Fanuc KAREL source: kt00972.KL

-- PROVISIONAL review KL for V770-1; original PC SHA256 310e2f795011a81680a6a24ac329b0ad1753ae2ed1f3e9ca645aaa79ceb5e1ae
-- Incomplete behavior may be omitted. Consult companion uncertainty JSON. Do not deploy.
PROGRAM KT00972
%NOLOCKGROUP
VAR
  ENTRY : INTEGER
  PNAME : STRING[80]
  VNAME : STRING[80]
  STATUS : INTEGER
-- UNRESOLVED_DECL VALUE type=002018
BEGIN
  -- UNRESOLVED_PC offsets 5-12; opcodes 9C,23
  -- UNRESOLVED_PC offsets 17-25; opcodes 3F,75
  -- UNRESOLVED_PC offsets 30-43; opcodes 3F,75
  -- UNRESOLVED_PC offsets 48-86; opcodes 27,22,22,2A,22,2A,22,22,B0
  -- UNRESOLVED_PC offsets 91-95; opcodes 7F
END KT00972
